// TIA Portal V17 export
// export: Created 2022-02-03T14:45:10.9428872Z, ExportSetting WithDefaults, DisplayName Totally Integrated Automation Portal, DisplayVersion V17, DisplayName TIA Portal Openness, DisplayVersion V17, DisplayName TIA Portal Version Control Interface, DisplayVersion V17, DisplayName SINAMICS Startdrive Advanced, DisplayVersion V17, DisplayName SINAMICS Startdrive G130, G150, S120, S150, SINAMICS MV, S210, DisplayVersion V17, DisplayName SINAMICS Startdrive G110M, G120, G120C, G120D, G120P, G115D, DisplayVersion V17, DisplayName STEP 7 Professional, DisplayVersion V17, DisplayName STEP 7 Safety, DisplayVersion V17, DisplayName WinCC Advanced, DisplayVersion V17
DATA_BLOCK "InstConveyor"   // DB4
VERSION : 0.1
// stored: Access Unpublished, AutoNumber true, DBAccessibleFromOPCUA true, DBAccessibleFromWebserver true, InstanceOfName Conveyor, InstanceOfType FB
"Conveyor"
   // VAR_INPUT
   //    operationMode : Bool;
   //    jogRight : Bool;
   //    jogLeft : Bool;
   //    conveyorIn : "typeConveyorInput";
   //    conveyorFault : Bool;
   //    weightOk : Bool;
   //    currentStoreFull : Bool;
   // END_VAR
   // VAR_OUTPUT
   //    conveyorRight : Bool;
   //    conveyorLeft : Bool;
   // END_VAR
   // VAR_IN_OUT
   //    occupiedBay : Array[1..3] of Bool;
   // END_VAR
   // VAR
   //    statAutoLeft : Bool;
   //    InstBayOccupied1 { S7_SetPoint := 'True'} : "BayOccupied";
   //    InstBayOccupied2 { S7_SetPoint := 'True'} : "BayOccupied";
   //    InstBayOccupied3 { S7_SetPoint := 'True'} : "BayOccupied";
   // END_VAR
BEGIN
END_DATA_BLOCK
